{attribute 'call_after_init'}
FUNCTION_BLOCK FB_AmphosAttenuatorEnable_Test EXTENDS FB_TestSuite
VAR_INPUT
END_VAR
VAR_OUTPUT
END_VAR
VAR
END_VAR

LocksWithHardwareFailure();
LocksWithLUTLeak();
LocksWithLOTAOLeak();
LocksWithLOCOLeak();
LocksWithMRC01Error();
LocksWhenAmphosOff();
EnablesWhenNoError();

METHOD EnablesWhenNoError
VAR
	stErrors : st_ErrorStates;
	bResult : BOOL;
END_VAR
TEST('EnablesWhenNoError');

bResult := F_AmphosAttenuatorEnable(bAmphosOn := TRUE, stErrors := stErrors);

AssertTrue(bResult, 'Amphos Attenuator should be enabled');

TEST_FINISHED();
END_METHOD

METHOD LocksWhenAmphosOff
VAR
	stErrors : st_ErrorStates;
	bResult : BOOL;
END_VAR
TEST('LocksWhenAmphosOff');

bResult := F_AmphosAttenuatorEnable(bAmphosOn := FALSE, stErrors := stErrors);

AssertFalse(bResult, 'Amphos Attenuator did not lock');

TEST_FINISHED();
END_METHOD

METHOD LocksWithHardwareFailure
VAR
	stErrors : st_ErrorStates;
	bResult : BOOL;
END_VAR
TEST('LocksWithHardwareFailure');

stErrors.bHardwareFailure := TRUE;
bResult := F_AmphosAttenuatorEnable(bAmphosOn := FALSE, stErrors := stErrors);

AssertFalse(bResult, 'Amphos Attenuator did not lock');

TEST_FINISHED();
END_METHOD

METHOD LocksWithLOCOLeak
VAR
	stErrors : st_ErrorStates;
	bResult : BOOL;
END_VAR
TEST('LocksWithLOCOLeak');

stErrors.bLeakOpcpaCarbideOn := TRUE;
bResult := F_AmphosAttenuatorEnable(bAmphosOn := TRUE, stErrors := stErrors);

AssertFalse(bResult, 'Amphos Attenuator did not lock');

TEST_FINISHED();
END_METHOD

METHOD LocksWithLOTAOLeak
VAR
	stErrors : st_ErrorStates;
	bResult : BOOL;
END_VAR
TEST('LocksWithLOTAOLeak');

stErrors.bLeakOpticalTableAmphosOn := TRUE;
bResult := F_AmphosAttenuatorEnable(bAmphosOn := TRUE, stErrors := stErrors);

AssertFalse(bResult, 'Amphos Attenuator did not lock');

TEST_FINISHED();
END_METHOD

METHOD LocksWithLUTLeak
VAR
	stErrors : st_ErrorStates;
	bResult : BOOL;
END_VAR
TEST('LocksWithLUTLeak');

stErrors.bLeakUnderTable := TRUE;
bResult := F_AmphosAttenuatorEnable(bAmphosOn := TRUE, stErrors := stErrors);

AssertFalse(bResult, 'Amphos Attenuator did not lock');

TEST_FINISHED();
END_METHOD

METHOD LocksWithMRC01Error
VAR
	stErrors : st_ErrorStates;
	bResult : BOOL;
END_VAR
TEST('LocksWithMRC01Error');

stErrors.bAmphosMRC01 := TRUE;
bResult := F_AmphosAttenuatorEnable(bAmphosOn := TRUE, stErrors := stErrors);

AssertFalse(bResult, 'Amphos Attenuator did not lock');

TEST_FINISHED();
END_METHOD

END_FUNCTION_BLOCK

(* stored: Version 1.1.0.1, ProductVersion 3.1.4022.17
   POU FB_AmphosAttenuatorEnable_Test: Id {56de8707-e9ed-440b-b040-6968f4b85d15}, SpecialFunc None
   Method EnablesWhenNoError: Id {e55da7b1-875b-41f3-8cfb-47fd92024193}
   Method LocksWhenAmphosOff: Id {7c2acb96-e983-4a47-9240-c6a18b5ecca6}
   Method LocksWithHardwareFailure: Id {7e58030a-eb57-4321-81e1-ea9542408654}
   Method LocksWithLOCOLeak: Id {27a899f8-27c4-4c8f-a19b-34716e76baff}
   Method LocksWithLOTAOLeak: Id {b04bb160-5174-43d1-8eaa-4d9b5223bc8d}
   Method LocksWithLUTLeak: Id {7c58bbfe-fca2-42a2-9b0c-f5516df547f9}
   Method LocksWithMRC01Error: Id {b0b2a6da-c52f-4e18-998e-104d429fd21d} *)
